// TwinCAT 3 PLC project TestProject
// ProgramVersion: 3.1.4020.4
// libraries:
//   Tc2_EtherCAT, * (Beckhoff Automation GmbH)
//   Tc2_MC2, * (Beckhoff Automation GmbH)
//   Tc2_Standard, * (Beckhoff Automation GmbH)
//   Tc2_System, * (Beckhoff Automation GmbH)
//   Tc3_Module, * (Beckhoff Automation GmbH)
//   tc_mca_std_lib, * (ESS)
// project tree:
//   DUTs/ ST_AxisHardware.TcDUT, ST_AxisParams.TcDUT, ST_EL7031CoEParams.TcDUT
//   / PlcTask.TcTTO
//   POUs/ FB_AxisConfig.TcPOU, FB_AxisEthMaster.TcPOU, FB_AxisHardware.TcPOU, FB_AxisRead5042.TcPOU, FB_AxisRead70x1.TcPOU, FB_AxisReadCoE.TcPOU, FB_AxisReadNC.TcPOU, FB_AxisReadParams.TcPOU, FB_AxisSetSlaveState.TcPOU, FB_AxisWrite5042.TcPOU, FB_AxisWrite70x1.TcPOU, FB_AxisWriteCoE.TcPOU, FB_AxisWriteNC.TcPOU, FB_AxisWriteParams.TcPOU, MAIN.TcPOU, FB_AxisMaster.TcPOU
// real-time tasks:
//   TASK PlcTask: cycle T#10ms, priority 20, ADS port 350
// motion (NC):
//   TASK NC-Task 1 SAF: cycle T#2ms, priority 4, ADS port 501
//   TASK NC-Task 1 SVB: cycle T#10ms, priority 8, ADS port 511
//   AXIS Axis 1 (id 1)
//     OtherSettings: AllowMotionCmdToSlave=true
//     encoder EncType=1
//     drive DrvType=5
//       TimeComp: TaskDelayCycles=1
//     controller CtrType=1
//       CtrPara: PriorControlFactor=1
//         Observer: BandWidth=20
//   AXIS Axis 2 (id 2)
//     OtherSettings: AllowMotionCmdToSlave=true
//     encoder EncType=29
//       EncPara: MaxCount=#xffffffff
//         Inc: RefSoftSyncMask=#x0000ffff
//     drive DrvType=24
//       TimeComp: TaskDelayCycles=1
//     controller CtrType=1
//       CtrPara: PriorControlFactor=1
//         Observer: BandWidth=20
//   AXIS Axis 3 (id 3)
//     OtherSettings: AllowMotionCmdToSlave=true
//     encoder EncType=29
//       EncPara: MaxCount=#xffffffff
//         Inc: RefSoftSyncMask=#x0000ffff
//     drive DrvType=24
//       TimeComp: TaskDelayCycles=1
//     controller CtrType=1
//       CtrPara: PriorControlFactor=1
//         Observer: BandWidth=20
// I/O:
//   DEVICE Device 1 (EtherCAT), AmsNetId 5.45.6.154.2.1
//     Term 1 (EK1200) [EK1200-5000 EtherCAT Power supply (2A E-Bus)]
//       Term 2 (EL7031) [EL7031 1Ch. Stepper motor output stage (24V, 1.5A)]
//       Term 3 (EL7041) [EL7041 1Ch. Stepper motor output stage (50V, 5A)]
//       Term 4 (EL5042) [EL5042 2Ch. BiSS-C Encoder]
//       Term 6 (EL1004) [EL1004 4Ch. Dig. Input 24V, 3ms]
//       Term 7 (EL1004) [EL1004 4Ch. Dig. Input 24V, 3ms]
//       Term 5 (EL9011) [EL9011 End Terminal]
// variable links:
//   (this object) <-> Device 1 (EtherCAT)/Term 1 (EK1200)/Term 2 (EL7031)
//     Drive/Inputs/In/nState1 @bit 3 <-> STM Status/Status/Error
//     Drive/Inputs/In/nState1 @bit 5 <-> STM Status/Status/Moving negative
//     Drive/Inputs/In/nState1 @bit 4 <-> STM Status/Status/Moving positive
//     Drive/Inputs/In/nState1 @bit 1 <-> STM Status/Status/Ready
//     Drive/Inputs/In/nState1 <-> STM Status/Status/Ready to enable
//     Drive/Inputs/In/nState1 @bit 6 <-> STM Status/Status/Torque reduced
//     Drive/Inputs/In/nState1 @bit 2 <-> STM Status/Status/Warning
//     Drive/Inputs/In/nState2 @bit 3 <-> STM Status/Status/Digital input 1
//     Drive/Inputs/In/nState2 @bit 4 <-> STM Status/Status/Digital input 2
//     Drive/Inputs/In/nState2 @bit 5 <-> STM Status/Status/Sync error
//     Drive/Inputs/In/nState2 @bit 7 <-> STM Status/Status/TxPDO Toggle
//     Drive/Inputs/In/nState4 @bit 1 <-> WcState/InputToggle
//     Drive/Inputs/In/nState4 <-> WcState/WcState
//     Drive/Outputs/Out/nCtrl1 <-> STM Control/Control/Enable
//     Drive/Outputs/Out/nCtrl1 @bit 2 <-> STM Control/Control/Reduce torque
//     Drive/Outputs/Out/nCtrl1 @bit 1 <-> STM Control/Control/Reset
//     Drive/Outputs/Out/nDataOut2[0] <-> STM Velocity/Velocity
//   (this object) <-> Device 1 (EtherCAT)/Term 1 (EK1200)/Term 4 (EL5042)
//     Enc/Inputs/In/nComState @bit 1 <-> WcState/InputToggle
//     Enc/Inputs/In/nComState <-> WcState/WcState
//     Enc/Inputs/In/nDataIn1 <-> FB Inputs Channel 1/Position
//     Enc/Inputs/In/nDataIn1 <-> FB Inputs Channel 2/Position
//     Enc/Inputs/In/nState1 @bit 12 <-> FB Inputs Channel 1/Status/Diag
//     Enc/Inputs/In/nState1 @bit 12 <-> FB Inputs Channel 2/Status/Diag
//     Enc/Inputs/In/nState1 @bit 1 <-> FB Inputs Channel 1/Status/Error
//     Enc/Inputs/In/nState1 @bit 1 <-> FB Inputs Channel 2/Status/Error
//     Enc/Inputs/In/nState1 @bit 14 <-> FB Inputs Channel 1/Status/Input cycle counter
//     Enc/Inputs/In/nState1 @bit 14 <-> FB Inputs Channel 2/Status/Input cycle counter
//     Enc/Inputs/In/nState1 @bit 2 <-> FB Inputs Channel 1/Status/Ready
//     Enc/Inputs/In/nState1 @bit 2 <-> FB Inputs Channel 2/Status/Ready
//     Enc/Inputs/In/nState1 @bit 13 <-> FB Inputs Channel 1/Status/TxPDO State
//     Enc/Inputs/In/nState1 @bit 13 <-> FB Inputs Channel 2/Status/TxPDO State
//     Enc/Inputs/In/nState1 <-> FB Inputs Channel 1/Status/Warning
//     Enc/Inputs/In/nState1 <-> FB Inputs Channel 2/Status/Warning
//   (this object) <-> Device 1 (EtherCAT)/Term 1 (EK1200)/Term 3 (EL7041)
//     Drive/Inputs/In/nState1 @bit 3 <-> STM Status/Status/Error
//     Drive/Inputs/In/nState1 @bit 5 <-> STM Status/Status/Moving negative
//     Drive/Inputs/In/nState1 @bit 4 <-> STM Status/Status/Moving positive
//     Drive/Inputs/In/nState1 @bit 1 <-> STM Status/Status/Ready
//     Drive/Inputs/In/nState1 <-> STM Status/Status/Ready to enable
//     Drive/Inputs/In/nState1 @bit 6 <-> STM Status/Status/Torque reduced
//     Drive/Inputs/In/nState1 @bit 2 <-> STM Status/Status/Warning
//     Drive/Inputs/In/nState2 @bit 3 <-> STM Status/Status/Digital input 1
//     Drive/Inputs/In/nState2 @bit 4 <-> STM Status/Status/Digital input 2
//     Drive/Inputs/In/nState4 @bit 1 <-> WcState/InputToggle
//     Drive/Inputs/In/nState4 <-> WcState/WcState
//     Drive/Outputs/Out/nCtrl1 <-> STM Control/Control/Enable
//     Drive/Outputs/Out/nCtrl1 @bit 2 <-> STM Control/Control/Reduce torque
//     Drive/Outputs/Out/nCtrl1 @bit 1 <-> STM Control/Control/Reset
//     Drive/Outputs/Out/nDataOut2[0] <-> STM Velocity/Velocity
//   TestProject Instance <-> Device 1 (EtherCAT)/Term 1 (EK1200)/Term 2 (EL7031)
//     PlcTask Inputs/MAIN.bLimitBwdM2 <-> STM Status/Status/Digital input 2
//     PlcTask Inputs/MAIN.bLimitFwdM2 <-> STM Status/Status/Digital input 1
//   TestProject Instance <-> Device 1 (EtherCAT)/Term 1 (EK1200)/Term 3 (EL7041)
//     PlcTask Inputs/MAIN.bLimitBwdM3 <-> STM Status/Status/Digital input 2
//     PlcTask Inputs/MAIN.bLimitFwdM3 <-> STM Status/Status/Digital input 1
//   TestProject Instance <-> Device 1 (EtherCAT)/Term 1 (EK1200)/Term 4 (EL5042)
//     PlcTask Inputs/MAIN.ams23Enc <-> InfoData/AdsAddr
//   TestProject Instance <-> NC-Task 1 SAF/Axes/Axis 1
//     PlcTask Inputs/MAIN.M1.fbLink.Axis.NcToPlc <-> Outputs/ToPlc
//     PlcTask Outputs/MAIN.M1.fbLink.Axis.PlcToNc <-> Inputs/FromPlc
//   TestProject Instance <-> NC-Task 1 SAF/Axes/Axis 2
//     PlcTask Inputs/MAIN.M2.fbLink.Axis.NcToPlc <-> Outputs/ToPlc
//     PlcTask Outputs/MAIN.M2.fbLink.Axis.PlcToNc <-> Inputs/FromPlc
//   TestProject Instance <-> NC-Task 1 SAF/Axes/Axis 3
//     PlcTask Inputs/MAIN.M3.fbLink.Axis.NcToPlc <-> Outputs/ToPlc
//     PlcTask Outputs/MAIN.M3.fbLink.Axis.PlcToNc <-> Inputs/FromPlc

CONFIGURATION TestProject
    RESOURCE PLC ON TwinCAT3
        TASK PlcTask(INTERVAL := T#10ms, PRIORITY := 20);
        PROGRAM MAIN WITH PlcTask : MAIN;
    END_RESOURCE
END_CONFIGURATION

// ---- DUTs/ST_AxisHardware.TcDUT
TYPE ST_AxisHardware :
STRUCT
	drive_type: UINT;
	enc_type: UINT;
	drive_ref: ST_DriveRef;
	enc_ref: ST_DriveRef;
END_STRUCT
END_TYPE

// ---- DUTs/ST_AxisParams.TcDUT
TYPE ST_AxisParams :
STRUCT
	unit: STRING := 'mm';
	ref_vel: LREAL;
	max_vel: LREAL;
	max_acc: LREAL := 15000;
	max_dec: LREAL := 15000;
	def_acc: LREAL := 1500;
	def_dec: LREAL := 1500;
	def_jerk: LREAL := 2250;
	home_search: LREAL;
	home_sync: LREAL;
	man_fast: LREAL;
	man_slow: LREAL;
	enable_min_soft_limit: BOOL;
	enable_max_soft_limit: BOOL;
	min_soft_limit: LREAL;
	max_soft_limit: LREAL;
	max_pos_lag_value: LREAL := 5;
	max_pos_lag_filter_time: LREAL := 0.02;
	dead_time: LREAL := 0.008;
	enc_scale: LREAL;
	enc_offset: LREAL;
	enc_invert: BOOL;
	mot_invert: BOOL;
	max_current: UINT;
	holding_current: UINT := 100;
	voltage: UINT := 24000;
	resistance: UINT := 100;
	emf: UINT := 0;
	full_steps: UINT := 200;
	speed_range: USINT := 1;
	enc_supply: USINT := 50;
	enc_clock: USINT := 9;
	enc_multi_bits: USINT := 0;
	enc_single_bits: USINT := 32;
END_STRUCT
END_TYPE

// ---- DUTs/ST_EL7031CoEParams.TcDUT
TYPE ST_EL7031CoEParams :
STRUCT
END_STRUCT
END_TYPE

// ---- POUs/MAIN.TcPOU
PROGRAM MAIN
VAR
	fbAxisEthMaster: FB_AxisEthMaster;
	M1: FB_AxisMaster;
	M2: FB_AxisMaster;
	M3: FB_AxisMaster;
	bFirstCycle: BOOL := TRUE;
END_VAR

// Set the initial configs
IF bFirstCycle THEN
	M2.stConfigSet.ref_vel := 10;
	M2.stConfigSet.max_vel := 20;
	M2.stConfigSet.man_fast := 15;
	M2.stConfigSet.man_slow := 5;
	M2.stConfigSet.enc_scale := 0.001;
	M2.stConfigSet.max_current := 1100;
	M3.stConfigSet.ref_vel := 11;
	M3.stConfigSet.max_vel := 21;
	M3.stConfigSet.man_fast := 16;
	M3.stConfigSet.man_slow := 6;
	M3.stConfigSet.enc_scale := 0.002;
	M3.stConfigSet.max_current := 1234;
	bFirstCycle := FALSE;
END_IF

// Bring MASTER to OP once SLAVEs are PRE-OP
fbAxisEthMaster(bExecute:=M1.bInitPreOp AND M2.bInitPreOp AND M3.bInitPreOp);

// Enable and pass Cfg
M1(bEnable:=TRUE,
	bInitCfg:=FALSE,
	bCfgRO:=FALSE,
	bUseLimits:=FALSE);
M2(bEnable:=TRUE,
	bInitCfg:=TRUE,
	bCfgRO:=FALSE,
	nEncCh:=1);
M3(bEnable:=TRUE,
	bInitCfg:=TRUE,
	bCfgRO:=TRUE,
	nEncCh:=2);

END_PROGRAM

// ---- POUs/FB_AxisEthMaster.TcPOU
FUNCTION_BLOCK FB_AxisEthMaster
VAR_INPUT
	bExecute: BOOL := TRUE;
END_VAR
VAR_OUTPUT
	bCfgReady: BOOL;
END_VAR
VAR
	amsNetID AT %I*: AMSNETID;
	fbMasterOp: FB_EcSetMasterState;
END_VAR

// Set master to OP
// This should wait until all relevant slaves are set to PREOP or they will be prematurely set to OP
fbMasterOp(sNetId:=F_CREATEAMSNETID(amsNetID),
	bExecute:=bExecute,
	reqState:=EC_DEVICE_STATE_OP);

END_FUNCTION_BLOCK

// ---- POUs/FB_AxisMaster.TcPOU
FUNCTION_BLOCK FB_AxisMaster
VAR_INPUT
	bEnable: BOOL;
	bInitCfg: BOOL := TRUE;
	bCfgRO: BOOL := FALSE;
	bUseLimits: BOOL;
	nEncCh: USINT;
END_VAR
VAR_OUTPUT
	bBrakeOut AT %I*: BOOL;
	bInitPreOp: BOOL;
	stConfigGet: ST_AxisParams;
END_VAR
VAR
	stConfigSet: ST_AxisParams;
	bLimitFwd AT %I*: BOOL;
	bLimitBwd AT %I*: BOOL;
	bHomeSensor AT %I*: BOOL;
	amsEncAddr AT %I*: AMSADDR;
	fbLink: FB_NcAxis;
	fbHardware: FB_AxisHardware;
	fbConfig: FB_AxisConfig;
	fbMasterGetOP: FB_EcGetMasterState;
	fbAxisSetOP: FB_AxisSetSlaveState;
	fbDrive: FB_DriveVirtual;
	stAxisStatus: DUT_AxisStatus_v0_01;
	bExecConfig: BOOL;
END_VAR

// Landing zone to link the AXIS_REF and update it
fbLink(En:=bEnable);
// Get terminal info
fbHardware(bExecute:=bEnable,
	Axis:=fbLink.Axis,
	amsEncAddr:=amsEncAddr,
	nEncCh:=nEncCh);
// If asked to initialize and we haven't, then initialize
IF bInitCfg AND NOT fbConfig.bInitDone THEN
	bExecConfig := TRUE;
// If read-only and not initializing, reject the write command
ELSIF bCfgRO THEN
	bExecConfig := FALSE;
// Otherwise, keep the value written over ADS
END_IF
// Read and/or write the config
fbConfig(bExecute:=bExecConfig AND fbHardware.bDone,
	stConfigSet:=stConfigSet,
	stHardware:=fbHardware.stHardware,
	Axis:=fbLink.Axis,
	bInitPreOp=>bInitPreOp,
	stConfigGet=>stConfigGet);
// Reset the execute bool
IF fbConfig.bDone AND NOT fbConfig.bError THEN
	bExecConfig := FALSE;
END_IF
// After the initial config is done, go to OP mode
// But first, make sure the master is in OP mode
IF fbConfig.bDone AND NOT fbConfig.bError AND fbMasterGetOP.state <> EC_DEVICE_STATE_OP THEN
	IF fbMasterGetOP.bExecute AND NOT fbMasterGetOP.bBusy THEN
		fbMasterGetOP.bExecute := FALSE;
	ELSE
		fbMasterGetOP.bExecute := TRUE;
	END_IF
END_IF
fbMasterGetOP(sNetId:=fbHardware.stHardware.drive_ref.sNetId);
fbAxisSetOP(bExecute:=fbConfig.bDone AND NOT fbConfig.bError,
	stHardware:=fbHardware.stHardware,
	reqState:=EC_DEVICE_STATE_OP);

// Disable brake while executing move **TODO** make this robust
bBrakeOut := fbDrive.bExecute;

IF NOT bUseLimits THEN
	bLimitFwd := TRUE;
	bLimitBwd := TRUE;
END_IF
// Execute incoming motion commands
fbDrive(En:=bEnable,
	bEnable:=bEnable AND fbConfig.bInitDone,
	bLimitFwd:=bLimitFwd,
	bLimitBwd:=bLimitBwd,
	bHomeSensor:=bHomeSensor,
	Axis:=fbLink.Axis);
stAxisStatus := fbDrive.stAxisStatus;
// Reset the execute bool
IF fbDrive.bDone AND NOT fbDrive.bError THEN
	fbDrive.bExecute := FALSE;
END_IF

END_FUNCTION_BLOCK

// ---- POUs/FB_AxisHardware.TcPOU
FUNCTION_BLOCK FB_AxisHardware
VAR_INPUT
	bExecute: BOOL;
	amsEncAddr: AMSADDR;
	nEncCh: USINT;
END_VAR
VAR_IN_OUT
	Axis: AXIS_REF;
END_VAR
VAR_OUTPUT
	bDone: BOOL;
	bBusy: BOOL;
	bError: BOOL;
	nErrorID: UDINT;
	stHardware: ST_AxisHardware;
END_VAR
VAR
	fbReadDriveAddress: MC_ReadDriveAddress;
	fbDriveId: FB_EcGetSlaveIdentity;
	fbEncId: FB_EcGetSlaveIdentity;
	fbADSRead: ADSREADEX;
	stDriveAddr: ST_DriveAddress;
	stDriveRef: ST_DriveRef;
	stEncRef: ST_DriveRef;
END_VAR

// Get drive ref using AXIS_REF
fbReadDriveAddress(Execute:=bExecute,
	Axis:=Axis,
	DriveAddress=>stDriveAddr);
stDriveRef.sNetId := stDriveAddr.NetID;
stDriveRef.nSlaveAddr := stDriveAddr.SlaveAddress;
stDriveRef.nDriveNo := stDriveAddr.Channel;
stHardware.drive_ref := stDriveRef;

// Get encoder ref using input args (cannot be derived from AXIS_REF)
stEncRef.sNetId := F_CreateAmsNetId(amsEncAddr.netId);
stEncRef.nSlaveAddr := amsEncAddr.port;
stEncRef.nDriveNo := nEncCh;
stHardware.enc_ref := stEncRef;

// Get the drive model (e.g. 7031)
IF stDriveRef.nSlaveAddr > 0 THEN
	fbDriveId(bExecute:=bExecute AND fbReadDriveAddress.Done,
		sNetId:=stDriveRef.sNetId,
		nSlaveAddr:=stDriveRef.nSlaveAddr);
	stHardware.drive_type := UDINT_TO_UINT(SHR(fbDriveID.identity.productCode, 16));
END_IF

// Get the encoder model (e.g. 5042)
IF stEncRef.nSlaveAddr > 0 THEN
	fbEncId(bExecute:=bExecute AND fbReadDriveAddress.Done,
		sNetId:=stEncRef.sNetId,
		nSlaveAddr:=stEncRef.nSlaveAddr);
	stHardware.enc_type := UDINT_TO_UINT(SHR(fbEncID.identity.productCode, 16));
END_IF

// Summarize outputs
bDone := fbReadDriveAddress.Done AND NOT fbDriveId.bBusy AND NOT fbEncId.bBusy;
bBusy := fbReadDriveAddress.Busy OR fbDriveId.bBusy OR fbEncId.bBusy;
bError := fbReadDriveAddress.Error OR fbDriveId.bError OR fbEncId.bError;
IF fbReadDriveAddress.ErrorID > 0 THEN
	nErrorID := fbReadDriveAddress.ErrorID;
ELSIF fbDriveId.nErrId >0 THEN
	nErrorID := fbDriveId.nErrId;
ELSE
	nErrorID := fbEncId.nErrId;
END_IF

END_FUNCTION_BLOCK

// ---- POUs/FB_AxisConfig.TcPOU
FUNCTION_BLOCK FB_AxisConfig
VAR_INPUT
	bExecute: BOOL; // Set, then get
	bExecGet: BOOL; // Only get
	bReset: BOOL;
	stConfigSet: ST_AxisParams;
	stHardware: ST_AxisHardware;
END_VAR
VAR_IN_OUT
	Axis: AXIS_REF;
END_VAR
VAR_OUTPUT
	bDone: BOOL;
	bValid: BOOL;
	bBusy: BOOL;
	bError: BOOL;
	nErrorID: UDINT;
	bInitDone: BOOL;
	bInitPreOp: BOOL;
	stConfigGet: ST_AxisParams;
END_VAR
VAR
	fbRead: FB_AxisReadParams;
	fbWrite: FB_AxisWriteParams;
	bDoRead: BOOL;
END_VAR

// Write first
fbWrite(bExecute:=bExecute,
	bReset:=bReset,
	stConfig:=stConfigSet,
	stHardware:=stHardware,
	Axis:=Axis,
	bInitPreOp=>bInitPreOp);
// Reset bDoRead if both execs are false
IF NOT bExecute AND NOT bExecGet THEN
	bDoRead := FALSE;
END_IF
// If bExecute is TRUE, wait untill after the write to read
IF bExecute THEN
	bDoRead := fbWrite.bDone;
ELSE
	bDoRead := bExecGet;
END_IF
// Notify that its ok to set master to OP.
// This block is really only used if we skip the write step.
IF bDoRead THEN
	bInitPreOP := TRUE;
END_IF
// Read now
fbRead(bExecute:=bDoRead,
	bReset:=bReset,
	stHardware:=stHardware,
	Axis:=Axis,
	stConfig=>stConfigGet,
	bValid=>bValid);
// Set the status outputs
bDone := fbWrite.bDone AND NOT fbRead.bBusy;
bBusy := fbWrite.bBusy OR fbRead.bBusy;
bError := fbWrite.bError OR fbRead.bError;
IF fbWrite.nErrorID > 0 THEN
	nErrorID := fbWrite.nErrorID;
ELSE
	nErrorID := fbRead.nErrorID;
END_IF
IF bDone THEN
	bInitDone := TRUE;
END_IF
IF bError THEN
	bInitDone := FALSE;
END_IF

END_FUNCTION_BLOCK

// ---- POUs/FB_AxisReadParams.TcPOU
FUNCTION_BLOCK FB_AxisReadParams
VAR_INPUT
	bExecute: BOOL;
	bReset: BOOL;
	stHardware: ST_AxisHardware;
END_VAR
VAR_OUTPUT
	stConfig: ST_AxisParams;
	bValid: BOOL;
	bBusy: BOOL;
	bError: BOOL;
	nErrorID: UDINT;
END_VAR
VAR_IN_OUT
	Axis: AXIS_REF;
END_VAR
VAR
	fbNCRead: FB_AxisReadNC;
	fbCoERead: FB_AxisReadCoE;
END_VAR

fbNCRead(bExecute:=bExecute,
	bReset:=bReset,
	stConfig:=stConfig,
	Axis:=Axis);
fbCoERead(bExecute:=bExecute,
	bReset:=bReset,
	stHardware:=stHardware,
	stConfig:=stConfig,
	Axis:=Axis);
bValid := fbNCRead.bValid AND NOT fbCoERead.bBusy AND NOT fbCoERead.bError AND bExecute;
bBusy := fbNCRead.bBusy OR fbCoERead.bBusy;
bError := fbNCRead.bError OR fbCoERead.bError;
IF fbNCRead.nErrorID > 0 THEN
	nErrorID := fbNCRead.nErrorID;
ELSE
	nErrorID := fbCoERead.nErrorID;
END_IF

END_FUNCTION_BLOCK

// ---- POUs/FB_AxisReadNC.TcPOU
FUNCTION_BLOCK FB_AxisReadNC
VAR_INPUT
	bExecute: BOOL;
	bReset: BOOL;
END_VAR
VAR_IN_OUT
	stConfig: ST_AxisParams;
	Axis: AXIS_REF;
END_VAR
VAR_OUTPUT
	bValid: BOOL;
	bBusy: BOOL;
	bError: BOOL;
	nErrorID: UDINT;
END_VAR
VAR
	fbReadRefVel: MC_ReadParameter;
  	fbReadRefVelRisingEdge: R_TRIG;
	fbReadMaxVel: MC_ReadParameter;
  	fbReadMaxVelRisingEdge: R_TRIG;
	fbReadMaxAcc: MC_ReadParameter;
  	fbReadMaxAccRisingEdge: R_TRIG;
	fbReadMaxDec: MC_ReadParameter;
  	fbReadMaxDecRisingEdge: R_TRIG;
	fbReadDefAcc: MC_ReadParameter;
  	fbReadDefAccRisingEdge: R_TRIG;
	fbReadDefDec: MC_ReadParameter;
  	fbReadDefDecRisingEdge: R_TRIG;
	fbReadDefJerk: MC_ReadParameter;
  	fbReadDefJerkRisingEdge: R_TRIG;
	fbReadHomeSearch: MC_ReadParameter;
  	fbReadHomeSearchRisingEdge: R_TRIG;
	fbReadHomeSync: MC_ReadParameter;
  	fbReadHomeSyncRisingEdge: R_TRIG;
	fbReadManFast: MC_ReadParameter;
  	fbReadManFastRisingEdge: R_TRIG;
	fbReadManSlow: MC_ReadParameter;
  	fbReadManSlowRisingEdge: R_TRIG;
	fbReadEnableMinSoftLimit: MC_ReadBoolParameter;
  	fbReadEnableMinSoftLimitRisingEdge: R_TRIG;
	fbReadEnableMaxSoftLimit: MC_ReadBoolParameter;
  	fbReadEnableMaxSoftLimitRisingEdge: R_TRIG;
	fbReadMinSoftLimit: MC_ReadParameter;
  	fbReadMinSoftLimitRisingEdge: R_TRIG;
	fbReadMaxSoftLimit: MC_ReadParameter;
  	fbReadMaxSoftLimitRisingEdge: R_TRIG;
	fbReadMaxPosLagValue: MC_ReadParameter;
  	fbReadMaxPosLagValueRisingEdge: R_TRIG;
	fbReadMaxPosLagFilterTime: MC_ReadParameter;
  	fbReadMaxPosLagFilterTimeRisingEdge: R_TRIG;
	fbReadDeadTime: MC_ReadParameter;
  	fbReadDeadTimeRisingEdge: R_TRIG;
	fbReadEncScale: MC_ReadParameter;
  	fbReadEncScaleRisingEdge: R_TRIG;
	fbReadEncOffset: MC_ReadParameter;
  	fbReadEncOffsetRisingEdge: R_TRIG;
	fbReadEncInvert: MC_ReadBoolParameter;
  	fbReadEncInvertRisingEdge: R_TRIG;
	fbReadMotInvert: MC_ReadBoolParameter;
  	fbReadMotInvertRisingEdge: R_TRIG;
END_VAR

// File auto-generated! Take care editing!
// Clears errors and allows a new read
IF bReset THEN
	bExecute := FALSE;
	bReset := FALSE;
END_IF
fbReadRefVel(Enable:=bExecute,
	ParameterNumber:=MC_AxisParameter.AxisRefVeloOnRefOutput,
	ReadMode:=E_ReadMode.READMODE_ONCE,
	Axis:=Axis);
fbReadRefVelRisingEdge(CLK:=fbReadRefVel.Valid AND NOT fbReadRefVel.Busy);
IF fbReadRefVelRisingEdge.Q AND NOT fbReadRefVel.Error THEN
	stConfig.ref_vel := fbReadRefVel.Value;
END_IF
fbReadMaxVel(Enable:=bExecute,
	ParameterNumber:=MC_AxisParameter.AxisMaxVelocity,
	ReadMode:=E_ReadMode.READMODE_ONCE,
	Axis:=Axis);
fbReadMaxVelRisingEdge(CLK:=fbReadMaxVel.Valid AND NOT fbReadMaxVel.Busy);
IF fbReadMaxVelRisingEdge.Q AND NOT fbReadMaxVel.Error THEN
	stConfig.max_vel := fbReadMaxVel.Value;
END_IF
fbReadMaxAcc(Enable:=bExecute,
	ParameterNumber:=MC_AxisParameter.MaxAccelerationSystem,
	ReadMode:=E_ReadMode.READMODE_ONCE,
	Axis:=Axis);
fbReadMaxAccRisingEdge(CLK:=fbReadMaxAcc.Valid AND NOT fbReadMaxAcc.Busy);
IF fbReadMaxAccRisingEdge.Q AND NOT fbReadMaxAcc.Error THEN
	stConfig.max_acc := fbReadMaxAcc.Value;
END_IF
fbReadMaxDec(Enable:=bExecute,
	ParameterNumber:=MC_AxisParameter.MaxDecelerationSystem,
	ReadMode:=E_ReadMode.READMODE_ONCE,
	Axis:=Axis);
fbReadMaxDecRisingEdge(CLK:=fbReadMaxDec.Valid AND NOT fbReadMaxDec.Busy);
IF fbReadMaxDecRisingEdge.Q AND NOT fbReadMaxDec.Error THEN
	stConfig.max_dec := fbReadMaxDec.Value;
END_IF
fbReadDefAcc(Enable:=bExecute,
	ParameterNumber:=MC_AxisParameter.AxisAcc,
	ReadMode:=E_ReadMode.READMODE_ONCE,
	Axis:=Axis);
fbReadDefAccRisingEdge(CLK:=fbReadDefAcc.Valid AND NOT fbReadDefAcc.Busy);
IF fbReadDefAccRisingEdge.Q AND NOT fbReadDefAcc.Error THEN
	stConfig.def_acc := fbReadDefAcc.Value;
END_IF
fbReadDefDec(Enable:=bExecute,
	ParameterNumber:=MC_AxisParameter.AxisDec,
	ReadMode:=E_ReadMode.READMODE_ONCE,
	Axis:=Axis);
fbReadDefDecRisingEdge(CLK:=fbReadDefDec.Valid AND NOT fbReadDefDec.Busy);
IF fbReadDefDecRisingEdge.Q AND NOT fbReadDefDec.Error THEN
	stConfig.def_dec := fbReadDefDec.Value;
END_IF
fbReadDefJerk(Enable:=bExecute,
	ParameterNumber:=MC_AxisParameter.AxisJerk,
	ReadMode:=E_ReadMode.READMODE_ONCE,
	Axis:=Axis);
fbReadDefJerkRisingEdge(CLK:=fbReadDefJerk.Valid AND NOT fbReadDefJerk.Busy);
IF fbReadDefJerkRisingEdge.Q AND NOT fbReadDefJerk.Error THEN
	stConfig.def_jerk := fbReadDefJerk.Value;
END_IF
fbReadHomeSearch(Enable:=bExecute,
	ParameterNumber:=MC_AxisParameter.AxisCalibrationVelocityForward,
	ReadMode:=E_ReadMode.READMODE_ONCE,
	Axis:=Axis);
fbReadHomeSearchRisingEdge(CLK:=fbReadHomeSearch.Valid AND NOT fbReadHomeSearch.Busy);
IF fbReadHomeSearchRisingEdge.Q AND NOT fbReadHomeSearch.Error THEN
	stConfig.home_search := fbReadHomeSearch.Value;
END_IF
fbReadHomeSync(Enable:=bExecute,
	ParameterNumber:=MC_AxisParameter.AxisCalibrationVelocityBackward,
	ReadMode:=E_ReadMode.READMODE_ONCE,
	Axis:=Axis);
fbReadHomeSyncRisingEdge(CLK:=fbReadHomeSync.Valid AND NOT fbReadHomeSync.Busy);
IF fbReadHomeSyncRisingEdge.Q AND NOT fbReadHomeSync.Error THEN
	stConfig.home_sync := fbReadHomeSync.Value;
END_IF
fbReadManFast(Enable:=bExecute,
	ParameterNumber:=MC_AxisParameter.AxisManualVelocityFast,
	ReadMode:=E_ReadMode.READMODE_ONCE,
	Axis:=Axis);
fbReadManFastRisingEdge(CLK:=fbReadManFast.Valid AND NOT fbReadManFast.Busy);
IF fbReadManFastRisingEdge.Q AND NOT fbReadManFast.Error THEN
	stConfig.man_fast := fbReadManFast.Value;
END_IF
fbReadManSlow(Enable:=bExecute,
	ParameterNumber:=MC_AxisParameter.AxisManualVelocitySlow,
	ReadMode:=E_ReadMode.READMODE_ONCE,
	Axis:=Axis);
fbReadManSlowRisingEdge(CLK:=fbReadManSlow.Valid AND NOT fbReadManSlow.Busy);
IF fbReadManSlowRisingEdge.Q AND NOT fbReadManSlow.Error THEN
	stConfig.man_slow := fbReadManSlow.Value;
END_IF
fbReadEnableMinSoftLimit(Enable:=bExecute,
	ParameterNumber:=MC_AxisParameter.EnableLimitNeg,
	ReadMode:=E_ReadMode.READMODE_ONCE,
	Axis:=Axis);
fbReadEnableMinSoftLimitRisingEdge(CLK:=fbReadEnableMinSoftLimit.Valid AND NOT fbReadEnableMinSoftLimit.Busy);
IF fbReadEnableMinSoftLimitRisingEdge.Q AND NOT fbReadEnableMinSoftLimit.Error THEN
	stConfig.enable_min_soft_limit := fbReadEnableMinSoftLimit.Value;
END_IF
fbReadEnableMaxSoftLimit(Enable:=bExecute,
	ParameterNumber:=MC_AxisParameter.EnableLimitPos,
	ReadMode:=E_ReadMode.READMODE_ONCE,
	Axis:=Axis);
fbReadEnableMaxSoftLimitRisingEdge(CLK:=fbReadEnableMaxSoftLimit.Valid AND NOT fbReadEnableMaxSoftLimit.Busy);
IF fbReadEnableMaxSoftLimitRisingEdge.Q AND NOT fbReadEnableMaxSoftLimit.Error THEN
	stConfig.enable_max_soft_limit := fbReadEnableMaxSoftLimit.Value;
END_IF
fbReadMinSoftLimit(Enable:=bExecute,
	ParameterNumber:=MC_AxisParameter.SWLimitNeg,
	ReadMode:=E_ReadMode.READMODE_ONCE,
	Axis:=Axis);
fbReadMinSoftLimitRisingEdge(CLK:=fbReadMinSoftLimit.Valid AND NOT fbReadMinSoftLimit.Busy);
IF fbReadMinSoftLimitRisingEdge.Q AND NOT fbReadMinSoftLimit.Error THEN
	stConfig.min_soft_limit := fbReadMinSoftLimit.Value;
END_IF
fbReadMaxSoftLimit(Enable:=bExecute,
	ParameterNumber:=MC_AxisParameter.SWLimitPos,
	ReadMode:=E_ReadMode.READMODE_ONCE,
	Axis:=Axis);
fbReadMaxSoftLimitRisingEdge(CLK:=fbReadMaxSoftLimit.Valid AND NOT fbReadMaxSoftLimit.Busy);
IF fbReadMaxSoftLimitRisingEdge.Q AND NOT fbReadMaxSoftLimit.Error THEN
	stConfig.max_soft_limit := fbReadMaxSoftLimit.Value;
END_IF
fbReadMaxPosLagValue(Enable:=bExecute,
	ParameterNumber:=MC_AxisParameter.MaxPositionLag,
	ReadMode:=E_ReadMode.READMODE_ONCE,
	Axis:=Axis);
fbReadMaxPosLagValueRisingEdge(CLK:=fbReadMaxPosLagValue.Valid AND NOT fbReadMaxPosLagValue.Busy);
IF fbReadMaxPosLagValueRisingEdge.Q AND NOT fbReadMaxPosLagValue.Error THEN
	stConfig.max_pos_lag_value := fbReadMaxPosLagValue.Value;
END_IF
fbReadMaxPosLagFilterTime(Enable:=bExecute,
	ParameterNumber:=MC_AxisParameter.AxisMaxPosLagFilterTime,
	ReadMode:=E_ReadMode.READMODE_ONCE,
	Axis:=Axis);
fbReadMaxPosLagFilterTimeRisingEdge(CLK:=fbReadMaxPosLagFilterTime.Valid AND NOT fbReadMaxPosLagFilterTime.Busy);
IF fbReadMaxPosLagFilterTimeRisingEdge.Q AND NOT fbReadMaxPosLagFilterTime.Error THEN
	stConfig.max_pos_lag_filter_time := fbReadMaxPosLagFilterTime.Value;
END_IF
fbReadDeadTime(Enable:=bExecute,
	ParameterNumber:=MC_AxisParameter.AxisDelayTimeVeloPosition,
	ReadMode:=E_ReadMode.READMODE_ONCE,
	Axis:=Axis);
fbReadDeadTimeRisingEdge(CLK:=fbReadDeadTime.Valid AND NOT fbReadDeadTime.Busy);
IF fbReadDeadTimeRisingEdge.Q AND NOT fbReadDeadTime.Error THEN
	stConfig.dead_time := fbReadDeadTime.Value;
END_IF
fbReadEncScale(Enable:=bExecute,
	ParameterNumber:=MC_AxisParameter.AxisEncoderScalingFactor,
	ReadMode:=E_ReadMode.READMODE_ONCE,
	Axis:=Axis);
fbReadEncScaleRisingEdge(CLK:=fbReadEncScale.Valid AND NOT fbReadEncScale.Busy);
IF fbReadEncScaleRisingEdge.Q AND NOT fbReadEncScale.Error THEN
	stConfig.enc_scale := fbReadEncScale.Value;
END_IF
fbReadEncOffset(Enable:=bExecute,
	ParameterNumber:=MC_AxisParameter.AxisEncoderOffset,
	ReadMode:=E_ReadMode.READMODE_ONCE,
	Axis:=Axis);
fbReadEncOffsetRisingEdge(CLK:=fbReadEncOffset.Valid AND NOT fbReadEncOffset.Busy);
IF fbReadEncOffsetRisingEdge.Q AND NOT fbReadEncOffset.Error THEN
	stConfig.enc_offset := fbReadEncOffset.Value;
END_IF
fbReadEncInvert(Enable:=bExecute,
	ParameterNumber:=MC_AxisParameter.AxisEncoderDirectionInverse,
	ReadMode:=E_ReadMode.READMODE_ONCE,
	Axis:=Axis);
fbReadEncInvertRisingEdge(CLK:=fbReadEncInvert.Valid AND NOT fbReadEncInvert.Busy);
IF fbReadEncInvertRisingEdge.Q AND NOT fbReadEncInvert.Error THEN
	stConfig.enc_invert := fbReadEncInvert.Value;
END_IF
fbReadMotInvert(Enable:=bExecute,
	ParameterNumber:=MC_AxisParameter.AxisMotorDirectionInverse,
	ReadMode:=E_ReadMode.READMODE_ONCE,
	Axis:=Axis);
fbReadMotInvertRisingEdge(CLK:=fbReadMotInvert.Valid AND NOT fbReadMotInvert.Busy);
IF fbReadMotInvertRisingEdge.Q AND NOT fbReadMotInvert.Error THEN
	stConfig.mot_invert := fbReadMotInvert.Value;
END_IF
bValid := fbReadRefVel.Valid AND fbReadMaxVel.Valid AND fbReadMaxAcc.Valid AND fbReadMaxDec.Valid AND fbReadDefAcc.Valid AND fbReadDefDec.Valid AND fbReadDefJerk.Valid AND fbReadHomeSearch.Valid AND fbReadHomeSync.Valid AND fbReadManFast.Valid AND fbReadManSlow.Valid AND fbReadEnableMinSoftLimit.Valid AND fbReadEnableMaxSoftLimit.Valid AND fbReadMinSoftLimit.Valid AND fbReadMaxSoftLimit.Valid AND fbReadMaxPosLagValue.Valid AND fbReadMaxPosLagFilterTime.Valid AND fbReadDeadTime.Valid AND fbReadEncScale.Valid AND fbReadEncOffset.Valid AND fbReadEncInvert.Valid AND fbReadMotInvert.Valid;
bBusy := fbReadRefVel.Busy OR fbReadMaxVel.Busy OR fbReadMaxAcc.Busy OR fbReadMaxDec.Busy OR fbReadDefAcc.Busy OR fbReadDefDec.Busy OR fbReadDefJerk.Busy OR fbReadHomeSearch.Busy OR fbReadHomeSync.Busy OR fbReadManFast.Busy OR fbReadManSlow.Busy OR fbReadEnableMinSoftLimit.Busy OR fbReadEnableMaxSoftLimit.Busy OR fbReadMinSoftLimit.Busy OR fbReadMaxSoftLimit.Busy OR fbReadMaxPosLagValue.Busy OR fbReadMaxPosLagFilterTime.Busy OR fbReadDeadTime.Busy OR fbReadEncScale.Busy OR fbReadEncOffset.Busy OR fbReadEncInvert.Busy OR fbReadMotInvert.Busy;
bError := fbReadRefVel.Error OR fbReadMaxVel.Error OR fbReadMaxAcc.Error OR fbReadMaxDec.Error OR fbReadDefAcc.Error OR fbReadDefDec.Error OR fbReadDefJerk.Error OR fbReadHomeSearch.Error OR fbReadHomeSync.Error OR fbReadManFast.Error OR fbReadManSlow.Error OR fbReadEnableMinSoftLimit.Error OR fbReadEnableMaxSoftLimit.Error OR fbReadMinSoftLimit.Error OR fbReadMaxSoftLimit.Error OR fbReadMaxPosLagValue.Error OR fbReadMaxPosLagFilterTime.Error OR fbReadDeadTime.Error OR fbReadEncScale.Error OR fbReadEncOffset.Error OR fbReadEncInvert.Error OR fbReadMotInvert.Error;
IF NOT bError THEN
	nErrorID := 0;
ELSIF fbReadRefVel.ErrorID > 0 THEN
	nErrorID := fbReadRefVel.ErrorID;
ELSIF fbReadMaxVel.ErrorID > 0 THEN
	nErrorID := fbReadMaxVel.ErrorID;
ELSIF fbReadMaxAcc.ErrorID > 0 THEN
	nErrorID := fbReadMaxAcc.ErrorID;
ELSIF fbReadMaxDec.ErrorID > 0 THEN
	nErrorID := fbReadMaxDec.ErrorID;
ELSIF fbReadDefAcc.ErrorID > 0 THEN
	nErrorID := fbReadDefAcc.ErrorID;
ELSIF fbReadDefDec.ErrorID > 0 THEN
	nErrorID := fbReadDefDec.ErrorID;
ELSIF fbReadDefJerk.ErrorID > 0 THEN
	nErrorID := fbReadDefJerk.ErrorID;
ELSIF fbReadHomeSearch.ErrorID > 0 THEN
	nErrorID := fbReadHomeSearch.ErrorID;
ELSIF fbReadHomeSync.ErrorID > 0 THEN
	nErrorID := fbReadHomeSync.ErrorID;
ELSIF fbReadManFast.ErrorID > 0 THEN
	nErrorID := fbReadManFast.ErrorID;
ELSIF fbReadManSlow.ErrorID > 0 THEN
	nErrorID := fbReadManSlow.ErrorID;
ELSIF fbReadEnableMinSoftLimit.ErrorID > 0 THEN
	nErrorID := fbReadEnableMinSoftLimit.ErrorID;
ELSIF fbReadEnableMaxSoftLimit.ErrorID > 0 THEN
	nErrorID := fbReadEnableMaxSoftLimit.ErrorID;
ELSIF fbReadMinSoftLimit.ErrorID > 0 THEN
	nErrorID := fbReadMinSoftLimit.ErrorID;
ELSIF fbReadMaxSoftLimit.ErrorID > 0 THEN
	nErrorID := fbReadMaxSoftLimit.ErrorID;
ELSIF fbReadMaxPosLagValue.ErrorID > 0 THEN
	nErrorID := fbReadMaxPosLagValue.ErrorID;
ELSIF fbReadMaxPosLagFilterTime.ErrorID > 0 THEN
	nErrorID := fbReadMaxPosLagFilterTime.ErrorID;
ELSIF fbReadDeadTime.ErrorID > 0 THEN
	nErrorID := fbReadDeadTime.ErrorID;
ELSIF fbReadEncScale.ErrorID > 0 THEN
	nErrorID := fbReadEncScale.ErrorID;
ELSIF fbReadEncOffset.ErrorID > 0 THEN
	nErrorID := fbReadEncOffset.ErrorID;
ELSIF fbReadEncInvert.ErrorID > 0 THEN
	nErrorID := fbReadEncInvert.ErrorID;
ELSIF fbReadMotInvert.ErrorID > 0 THEN
	nErrorID := fbReadMotInvert.ErrorID;
END_IF

END_FUNCTION_BLOCK

// ---- POUs/FB_AxisReadCoE.TcPOU
FUNCTION_BLOCK FB_AxisReadCoE
VAR_INPUT
	bExecute: BOOL;
	bReset: BOOL;
	stHardware: ST_AxisHardware;
END_VAR
VAR_IN_OUT
	stConfig: ST_AxisParams;
	Axis: AXIS_REF;
END_VAR
VAR_OUTPUT
	bBusy: BOOL;
	bError: BOOL;
	nErrorID: UDINT;
END_VAR
VAR
	fbRead70x1: FB_AxisRead70x1;
	fbRead5042: FB_AxisRead5042;
	bBusyDrive: BOOL;
	bBusyEnc: BOOL;
	bErrorDrive: BOOL;
	bErrorEnc: BOOL;
	iErrorDriveADS: UDINT;
	iErrorEncADS: UDINT;
	iErrorDriveCAN: UDINT;
	iErrorEncCAN: UDINT;
END_VAR

CASE stHardware.drive_type OF
	0:
		bBusyDrive := FALSE;
		bErrorDrive := FALSE;
		iErrorDriveAds := 0;
		iErrorDriveCAN := 0;
	7031, 7041:
		fbRead70x1(bExecute:=bExecute,
			bReset:=bReset,
			stDriveRef:=stHardware.drive_ref,
			stConfig:=stConfig,
			Axis:=Axis,
			bBusy=>bBusyDrive,
			bError=>bErrorDrive,
			iAdsErrId=>iErrorDriveAds,
			iCANopenErrId=>iErrorDriveCAN);
	ELSE
		bBusyDrive := FALSE;
		bErrorDrive := TRUE;
		iErrorDriveAds := 1;
		iErrorDriveCAN := 0;
END_CASE
CASE stHardware.enc_type OF
	0:
		bBusyEnc := FALSE;
		bErrorEnc := FALSE;
		iErrorEncAds := 0;
		iErrorEncCAN := 0;
	5042:
		fbRead5042(bExecute:=bExecute,
			bReset:=bReset,
			stDriveRef:=stHardware.enc_ref,
			stConfig:=stConfig,
			Axis:=Axis,
			bBusy=>bBusyEnc,
			bError=>bErrorEnc,
			iAdsErrId=>iErrorEncAds,
			iCANopenErrId=>iErrorEncCAN);
	ELSE
		bBusyEnc := FALSE;
		bErrorEnc := TRUE;
		iErrorEncAds := 1;
		iErrorEncCAN := 0;
END_CASE
bBusy := bBusyDrive OR bBusyEnc;
bError := bErrorDrive OR bErrorEnc;
IF iErrorDriveAds > 0 THEN
	nErrorID := iErrorDriveAds;
ELSIF iErrorDriveCAN > 0 THEN
	nErrorID := iErrorDriveCAN;
ELSIF iErrorEncAds > 0 THEN
	nErrorID := iErrorEncAds;
ELSE
	nErrorID := iErrorEncCAN;
END_IF

END_FUNCTION_BLOCK

// ---- POUs/FB_AxisRead70x1.TcPOU
FUNCTION_BLOCK FB_AxisRead70x1
VAR_INPUT
	bExecute: BOOL;
	bReset: BOOL;
	stDriveRef: ST_DriveRef;
END_VAR
VAR_IN_OUT
	stConfig: ST_AxisParams;
	Axis: AXIS_REF;
END_VAR
VAR_OUTPUT
	bBusy: BOOL;
	bError: BOOL;
	iAdsErrId: UINT;
	iCANopenErrId: UINT;
END_VAR
VAR
	fbReadMaxCurrent: FB_CoERead_ByDriveRef;
	nIndMaxCurrent: WORD;
	fbReadHoldingCurrent: FB_CoERead_ByDriveRef;
	nIndHoldingCurrent: WORD;
	fbReadVoltage: FB_CoERead_ByDriveRef;
	nIndVoltage: WORD;
	fbReadResistance: FB_CoERead_ByDriveRef;
	nIndResistance: WORD;
	fbReadEmf: FB_CoERead_ByDriveRef;
	nIndEmf: WORD;
	fbReadFullSteps: FB_CoERead_ByDriveRef;
	nIndFullSteps: WORD;
	fbReadSpeedRange: FB_CoERead_ByDriveRef;
	nIndSpeedRange: WORD;
END_VAR

// File auto-generated! Take care editing!
// Clears errors and allows a new read
IF bReset THEN
	bExecute := FALSE;
	bReset := FALSE;
END_IF
nIndMaxCurrent := 16#8010;
fbReadMaxCurrent(bExecute:=bExecute,
	stDriveRef:=stDriveRef,
	nindex:=nIndMaxCurrent,
	nSubIndex:=16#01,
	pDstBuf:=ADR(stConfig.max_current),
	cbBufLen:=SIZEOF(stConfig.max_current));
nIndHoldingCurrent := 16#8010;
fbReadHoldingCurrent(bExecute:=bExecute,
	stDriveRef:=stDriveRef,
	nindex:=nIndHoldingCurrent,
	nSubIndex:=16#02,
	pDstBuf:=ADR(stConfig.holding_current),
	cbBufLen:=SIZEOF(stConfig.holding_current));
nIndVoltage := 16#8010;
fbReadVoltage(bExecute:=bExecute,
	stDriveRef:=stDriveRef,
	nindex:=nIndVoltage,
	nSubIndex:=16#03,
	pDstBuf:=ADR(stConfig.voltage),
	cbBufLen:=SIZEOF(stConfig.voltage));
nIndResistance := 16#8010;
fbReadResistance(bExecute:=bExecute,
	stDriveRef:=stDriveRef,
	nindex:=nIndResistance,
	nSubIndex:=16#04,
	pDstBuf:=ADR(stConfig.resistance),
	cbBufLen:=SIZEOF(stConfig.resistance));
nIndEmf := 16#8010;
fbReadEmf(bExecute:=bExecute,
	stDriveRef:=stDriveRef,
	nindex:=nIndEmf,
	nSubIndex:=16#05,
	pDstBuf:=ADR(stConfig.emf),
	cbBufLen:=SIZEOF(stConfig.emf));
nIndFullSteps := 16#8010;
fbReadFullSteps(bExecute:=bExecute,
	stDriveRef:=stDriveRef,
	nindex:=nIndFullSteps,
	nSubIndex:=16#06,
	pDstBuf:=ADR(stConfig.full_steps),
	cbBufLen:=SIZEOF(stConfig.full_steps));
nIndSpeedRange := 16#8012;
fbReadSpeedRange(bExecute:=bExecute,
	stDriveRef:=stDriveRef,
	nindex:=nIndSpeedRange,
	nSubIndex:=16#05,
	pDstBuf:=ADR(stConfig.speed_range),
	cbBufLen:=SIZEOF(stConfig.speed_range));
bBusy := fbReadMaxCurrent.bBusy OR fbReadHoldingCurrent.bBusy OR fbReadVoltage.bBusy OR fbReadResistance.bBusy OR fbReadEmf.bBusy OR fbReadFullSteps.bBusy OR fbReadSpeedRange.bBusy;
bError := fbReadMaxCurrent.bError OR fbReadHoldingCurrent.bError OR fbReadVoltage.bError OR fbReadResistance.bError OR fbReadEmf.bError OR fbReadFullSteps.bError OR fbReadSpeedRange.bError;
IF NOT bError THEN
	iAdsErrId := 0;
ELSIF fbReadMaxCurrent.iAdsErrId > 0 THEN
	iAdsErrId := fbReadMaxCurrent.iAdsErrId;
ELSIF fbReadHoldingCurrent.iAdsErrId > 0 THEN
	iAdsErrId := fbReadHoldingCurrent.iAdsErrId;
ELSIF fbReadVoltage.iAdsErrId > 0 THEN
	iAdsErrId := fbReadVoltage.iAdsErrId;
ELSIF fbReadResistance.iAdsErrId > 0 THEN
	iAdsErrId := fbReadResistance.iAdsErrId;
ELSIF fbReadEmf.iAdsErrId > 0 THEN
	iAdsErrId := fbReadEmf.iAdsErrId;
ELSIF fbReadFullSteps.iAdsErrId > 0 THEN
	iAdsErrId := fbReadFullSteps.iAdsErrId;
ELSIF fbReadSpeedRange.iAdsErrId > 0 THEN
	iAdsErrId := fbReadSpeedRange.iAdsErrId;
END_IF
IF NOT bError THEN
	iCANopenErrId := 0;
ELSIF fbReadMaxCurrent.iCANopenErrId > 0 THEN
	iCANopenErrId := fbReadMaxCurrent.iCANopenErrId;
ELSIF fbReadHoldingCurrent.iCANopenErrId > 0 THEN
	iCANopenErrId := fbReadHoldingCurrent.iCANopenErrId;
ELSIF fbReadVoltage.iCANopenErrId > 0 THEN
	iCANopenErrId := fbReadVoltage.iCANopenErrId;
ELSIF fbReadResistance.iCANopenErrId > 0 THEN
	iCANopenErrId := fbReadResistance.iCANopenErrId;
ELSIF fbReadEmf.iCANopenErrId > 0 THEN
	iCANopenErrId := fbReadEmf.iCANopenErrId;
ELSIF fbReadFullSteps.iCANopenErrId > 0 THEN
	iCANopenErrId := fbReadFullSteps.iCANopenErrId;
ELSIF fbReadSpeedRange.iCANopenErrId > 0 THEN
	iCANopenErrId := fbReadSpeedRange.iCANopenErrId;
END_IF

END_FUNCTION_BLOCK

// ---- POUs/FB_AxisRead5042.TcPOU
FUNCTION_BLOCK FB_AxisRead5042
VAR_INPUT
	bExecute: BOOL;
	bReset: BOOL;
	stDriveRef: ST_DriveRef;
END_VAR
VAR_IN_OUT
	stConfig: ST_AxisParams;
	Axis: AXIS_REF;
END_VAR
VAR_OUTPUT
	bBusy: BOOL;
	bError: BOOL;
	iAdsErrId: UINT;
	iCANopenErrId: UINT;
END_VAR
VAR
	fbReadEncSupply: FB_CoERead_ByDriveRef;
	nIndEncSupply: WORD;
	fbReadEncClock: FB_CoERead_ByDriveRef;
	nIndEncClock: WORD;
	fbReadEncMultiBits: FB_CoERead_ByDriveRef;
	nIndEncMultiBits: WORD;
	fbReadEncSingleBits: FB_CoERead_ByDriveRef;
	nIndEncSingleBits: WORD;
END_VAR

// File auto-generated! Take care editing!
// Clears errors and allows a new read
IF bReset THEN
	bExecute := FALSE;
	bReset := FALSE;
END_IF
nIndEncSupply := 16#8008;
fbReadEncSupply(bExecute:=bExecute,
	stDriveRef:=stDriveRef,
	nindex:=nIndEncSupply,
	nSubIndex:=16#12,
	pDstBuf:=ADR(stConfig.enc_supply),
	cbBufLen:=SIZEOF(stConfig.enc_supply));
CASE stDriveRef.nDriveNo OF
	1:
		nIndEncClock := 16#8008;
	2:
		nIndEncClock := 16#8018;
END_CASE
fbReadEncClock(bExecute:=bExecute,
	stDriveRef:=stDriveRef,
	nindex:=nIndEncClock,
	nSubIndex:=16#13,
	pDstBuf:=ADR(stConfig.enc_clock),
	cbBufLen:=SIZEOF(stConfig.enc_clock));
CASE stDriveRef.nDriveNo OF
	1:
		nIndEncMultiBits := 16#8008;
	2:
		nIndEncMultiBits := 16#8018;
END_CASE
fbReadEncMultiBits(bExecute:=bExecute,
	stDriveRef:=stDriveRef,
	nindex:=nIndEncMultiBits,
	nSubIndex:=16#15,
	pDstBuf:=ADR(stConfig.enc_multi_bits),
	cbBufLen:=SIZEOF(stConfig.enc_multi_bits));
CASE stDriveRef.nDriveNo OF
	1:
		nIndEncSingleBits := 16#8008;
	2:
		nIndEncSingleBits := 16#8018;
END_CASE
fbReadEncSingleBits(bExecute:=bExecute,
	stDriveRef:=stDriveRef,
	nindex:=nIndEncSingleBits,
	nSubIndex:=16#16,
	pDstBuf:=ADR(stConfig.enc_single_bits),
	cbBufLen:=SIZEOF(stConfig.enc_single_bits));
bBusy := fbReadEncSupply.bBusy OR fbReadEncClock.bBusy OR fbReadEncMultiBits.bBusy OR fbReadEncSingleBits.bBusy;
bError := fbReadEncSupply.bError OR fbReadEncClock.bError OR fbReadEncMultiBits.bError OR fbReadEncSingleBits.bError;
IF NOT bError THEN
	iAdsErrId := 0;
ELSIF fbReadEncSupply.iAdsErrId > 0 THEN
	iAdsErrId := fbReadEncSupply.iAdsErrId;
ELSIF fbReadEncClock.iAdsErrId > 0 THEN
	iAdsErrId := fbReadEncClock.iAdsErrId;
ELSIF fbReadEncMultiBits.iAdsErrId > 0 THEN
	iAdsErrId := fbReadEncMultiBits.iAdsErrId;
ELSIF fbReadEncSingleBits.iAdsErrId > 0 THEN
	iAdsErrId := fbReadEncSingleBits.iAdsErrId;
END_IF
IF NOT bError THEN
	iCANopenErrId := 0;
ELSIF fbReadEncSupply.iCANopenErrId > 0 THEN
	iCANopenErrId := fbReadEncSupply.iCANopenErrId;
ELSIF fbReadEncClock.iCANopenErrId > 0 THEN
	iCANopenErrId := fbReadEncClock.iCANopenErrId;
ELSIF fbReadEncMultiBits.iCANopenErrId > 0 THEN
	iCANopenErrId := fbReadEncMultiBits.iCANopenErrId;
ELSIF fbReadEncSingleBits.iCANopenErrId > 0 THEN
	iCANopenErrId := fbReadEncSingleBits.iCANopenErrId;
END_IF

END_FUNCTION_BLOCK

// ---- POUs/FB_AxisWriteParams.TcPOU
FUNCTION_BLOCK FB_AxisWriteParams
VAR_INPUT
	bExecute: BOOL;
	bReset: BOOL;
	stConfig: ST_AxisParams;
	stHardware: ST_AxisHardware;
END_VAR
VAR_IN_OUT
	Axis: AXIS_REF;
END_VAR
VAR_OUTPUT
	bInitPreOp: BOOL;
	bDone: BOOL;
	bBusy: BOOL;
	bError: BOOL;
	nErrorID: UDINT;
END_VAR
VAR
	bDoWrite: BOOL;
	fbNCWrite: FB_AxisWriteNC;
	fbCoEWrite: FB_AxisWriteCoE;
	fbPrepWrite: FB_AxisSetSlaveState;
	fbInitState: FB_AxisSetSlaveState;
	fbPreOpState: FB_AxisSetSlaveState;
END_VAR

// Do not write unless axis is disabled. Leave TRUE after done to avoid resetting errors, etc.
bDoWrite := bExecute AND (Axis.Status.MotionState = MC_AXISSTATE_DISABLED OR bDone);
// Move to PREOP to prepare for writing
fbPrepWrite(bExecute:=bDoWrite,
	stHardware:=stHardware,
	reqState:=EC_DEVICE_STATE_PREOP);
// The first time we're here, report that we've set to PREOP so master can move to OP
IF fbPrepWrite.bDone AND NOT fbPrepWrite.bError THEN
	bInitPreOP := TRUE;
END_IF
// Do the write
fbNCWrite(bExecute:=fbPrepWrite.bDone AND NOT fbPrepWrite.bError,
	bReset:=bReset,
	stConfig:=stConfig,
	Axis:=Axis);
fbCoEWrite(bExecute:=fbNCWrite.bExecute,
	bReset:=bReset,
	stHardware:=stHardware,
	stConfig:=stConfig,
	Axis:=Axis);
// Move to INIT and back to PRE-OP for params that need a full restart
fbInitState(bExecute:=fbNCWrite.bDone AND NOT fbNCWrite.bError AND fbCoEWrite.bBusy AND NOT fbCoEWrite.bError,
	stHardware:=stHardware,
	reqState:=EC_DEVICE_STATE_INIT);
fbPreOpState(bExecute:=fbInitState.bDone AND NOT fbInitState.bError,
	stHardware:=stHardware,
	reqSTate:=EC_DEVICE_STATE_PREOP);
bDone := fbPreOpState.bDone;
bBusy := fbNCWrite.bBusy OR fbCoEWrite.bBusy OR fbPrepWrite.bBusy OR fbInitState.bBusy OR fbPreOpState.bBusy;
bError := fbNCWrite.bError OR fbCoEWrite.bError OR fbPrepWrite.bError OR fbInitState.bError OR fbPreOpState.bError;
IF fbNCWrite.nErrorID > 0 THEN
	nErrorID := fbNCWrite.nErrorID;
ELSIF fbCoeWrite.nErrorID > 0 THEN
	nErrorID := fbCoEWrite.nErrorID;
ELSIF fbPrepWrite.nErrId > 0 THEN
	nErrorID := fbPrepWrite.nErrId;
ELSIF fbInitSTate.nErrId > 0 THEN
	nErrorID := fbInitState.nErrId;
ELSE
	nErrorID := fbPreOpState.nErrId;
END_IF

END_FUNCTION_BLOCK

// ---- POUs/FB_AxisWriteNC.TcPOU
FUNCTION_BLOCK FB_AxisWriteNC
VAR_INPUT
	bExecute: BOOL;
	bReset: BOOL;
END_VAR
VAR_IN_OUT
	stConfig: ST_AxisParams;
	Axis: AXIS_REF;
END_VAR
VAR_OUTPUT
	bDone: BOOL;
	bBusy: BOOL;
	bError: BOOL;
	nErrorID: UDINT;
END_VAR
VAR
	fbWriteRefVel: MC_WriteParameter;
	fbWriteMaxVel: MC_WriteParameter;
	fbWriteMaxAcc: MC_WriteParameter;
	fbWriteMaxDec: MC_WriteParameter;
	fbWriteDefAcc: MC_WriteParameter;
	fbWriteDefDec: MC_WriteParameter;
	fbWriteDefJerk: MC_WriteParameter;
	fbWriteHomeSearch: MC_WriteParameter;
	fbWriteHomeSync: MC_WriteParameter;
	fbWriteManFast: MC_WriteParameter;
	fbWriteManSlow: MC_WriteParameter;
	fbWriteEnableMinSoftLimit: MC_WriteBoolParameter;
	fbWriteEnableMaxSoftLimit: MC_WriteBoolParameter;
	fbWriteMinSoftLimit: MC_WriteParameter;
	fbWriteMaxSoftLimit: MC_WriteParameter;
	fbWriteMaxPosLagValue: MC_WriteParameter;
	fbWriteMaxPosLagFilterTime: MC_WriteParameter;
	fbWriteDeadTime: MC_WriteParameter;
	fbWriteEncScale: MC_WriteParameter;
	fbWriteEncOffset: MC_WriteParameter;
	fbWriteEncInvert: MC_WriteBoolParameter;
	fbWriteMotInvert: MC_WriteBoolParameter;
END_VAR

// File auto-generated! Take care editing!
// Clears errors and allows a new read
IF bReset THEN
	bExecute := FALSE;
	bReset := FALSE;
END_IF
fbWriteRefVel(Execute:=bExecute,
	ParameterNumber:=MC_AxisParameter.AxisRefVeloOnRefOutput,
	Value:=stConfig.ref_vel,
	Axis:=Axis);
fbWriteMaxVel(Execute:=bExecute,
	ParameterNumber:=MC_AxisParameter.AxisMaxVelocity,
	Value:=stConfig.max_vel,
	Axis:=Axis);
fbWriteMaxAcc(Execute:=bExecute,
	ParameterNumber:=MC_AxisParameter.MaxAccelerationSystem,
	Value:=stConfig.max_acc,
	Axis:=Axis);
fbWriteMaxDec(Execute:=bExecute,
	ParameterNumber:=MC_AxisParameter.MaxDecelerationSystem,
	Value:=stConfig.max_dec,
	Axis:=Axis);
fbWriteDefAcc(Execute:=bExecute,
	ParameterNumber:=MC_AxisParameter.AxisAcc,
	Value:=stConfig.def_acc,
	Axis:=Axis);
fbWriteDefDec(Execute:=bExecute,
	ParameterNumber:=MC_AxisParameter.AxisDec,
	Value:=stConfig.def_dec,
	Axis:=Axis);
fbWriteDefJerk(Execute:=bExecute,
	ParameterNumber:=MC_AxisParameter.AxisJerk,
	Value:=stConfig.def_jerk,
	Axis:=Axis);
fbWriteHomeSearch(Execute:=bExecute,
	ParameterNumber:=MC_AxisParameter.AxisCalibrationVelocityForward,
	Value:=stConfig.home_search,
	Axis:=Axis);
fbWriteHomeSync(Execute:=bExecute,
	ParameterNumber:=MC_AxisParameter.AxisCalibrationVelocityBackward,
	Value:=stConfig.home_sync,
	Axis:=Axis);
fbWriteManFast(Execute:=bExecute,
	ParameterNumber:=MC_AxisParameter.AxisManualVelocityFast,
	Value:=stConfig.man_fast,
	Axis:=Axis);
fbWriteManSlow(Execute:=bExecute,
	ParameterNumber:=MC_AxisParameter.AxisManualVelocitySlow,
	Value:=stConfig.man_slow,
	Axis:=Axis);
fbWriteEnableMinSoftLimit(Execute:=bExecute,
	ParameterNumber:=MC_AxisParameter.EnableLimitNeg,
	Value:=stConfig.enable_min_soft_limit,
	Axis:=Axis);
fbWriteEnableMaxSoftLimit(Execute:=bExecute,
	ParameterNumber:=MC_AxisParameter.EnableLimitPos,
	Value:=stConfig.enable_max_soft_limit,
	Axis:=Axis);
fbWriteMinSoftLimit(Execute:=bExecute,
	ParameterNumber:=MC_AxisParameter.SWLimitNeg,
	Value:=stConfig.min_soft_limit,
	Axis:=Axis);
fbWriteMaxSoftLimit(Execute:=bExecute,
	ParameterNumber:=MC_AxisParameter.SWLimitPos,
	Value:=stConfig.max_soft_limit,
	Axis:=Axis);
fbWriteMaxPosLagValue(Execute:=bExecute,
	ParameterNumber:=MC_AxisParameter.MaxPositionLag,
	Value:=stConfig.max_pos_lag_value,
	Axis:=Axis);
fbWriteMaxPosLagFilterTime(Execute:=bExecute,
	ParameterNumber:=MC_AxisParameter.AxisMaxPosLagFilterTime,
	Value:=stConfig.max_pos_lag_filter_time,
	Axis:=Axis);
fbWriteDeadTime(Execute:=bExecute,
	ParameterNumber:=MC_AxisParameter.AxisDelayTimeVeloPosition,
	Value:=stConfig.dead_time,
	Axis:=Axis);
fbWriteEncScale(Execute:=bExecute,
	ParameterNumber:=MC_AxisParameter.AxisEncoderScalingFactor,
	Value:=stConfig.enc_scale,
	Axis:=Axis);
fbWriteEncOffset(Execute:=bExecute,
	ParameterNumber:=MC_AxisParameter.AxisEncoderOffset,
	Value:=stConfig.enc_offset,
	Axis:=Axis);
fbWriteEncInvert(Execute:=bExecute,
	ParameterNumber:=MC_AxisParameter.AxisEncoderDirectionInverse,
	Value:=stConfig.enc_invert,
	Axis:=Axis);
fbWriteMotInvert(Execute:=bExecute,
	ParameterNumber:=MC_AxisParameter.AxisMotorDirectionInverse,
	Value:=stConfig.mot_invert,
	Axis:=Axis);
bDone := fbWriteRefVel.Done AND fbWriteMaxVel.Done AND fbWriteMaxAcc.Done AND fbWriteMaxDec.Done AND fbWriteDefAcc.Done AND fbWriteDefDec.Done AND fbWriteDefJerk.Done AND fbWriteHomeSearch.Done AND fbWriteHomeSync.Done AND fbWriteManFast.Done AND fbWriteManSlow.Done AND fbWriteEnableMinSoftLimit.Done AND fbWriteEnableMaxSoftLimit.Done AND fbWriteMinSoftLimit.Done AND fbWriteMaxSoftLimit.Done AND fbWriteMaxPosLagValue.Done AND fbWriteMaxPosLagFilterTime.Done AND fbWriteDeadTime.Done AND fbWriteEncScale.Done AND fbWriteEncOffset.Done AND fbWriteEncInvert.Done AND fbWriteMotInvert.Done;
bBusy := fbWriteRefVel.Busy OR fbWriteMaxVel.Busy OR fbWriteMaxAcc.Busy OR fbWriteMaxDec.Busy OR fbWriteDefAcc.Busy OR fbWriteDefDec.Busy OR fbWriteDefJerk.Busy OR fbWriteHomeSearch.Busy OR fbWriteHomeSync.Busy OR fbWriteManFast.Busy OR fbWriteManSlow.Busy OR fbWriteEnableMinSoftLimit.Busy OR fbWriteEnableMaxSoftLimit.Busy OR fbWriteMinSoftLimit.Busy OR fbWriteMaxSoftLimit.Busy OR fbWriteMaxPosLagValue.Busy OR fbWriteMaxPosLagFilterTime.Busy OR fbWriteDeadTime.Busy OR fbWriteEncScale.Busy OR fbWriteEncOffset.Busy OR fbWriteEncInvert.Busy OR fbWriteMotInvert.Busy;
bError := fbWriteRefVel.Error OR fbWriteMaxVel.Error OR fbWriteMaxAcc.Error OR fbWriteMaxDec.Error OR fbWriteDefAcc.Error OR fbWriteDefDec.Error OR fbWriteDefJerk.Error OR fbWriteHomeSearch.Error OR fbWriteHomeSync.Error OR fbWriteManFast.Error OR fbWriteManSlow.Error OR fbWriteEnableMinSoftLimit.Error OR fbWriteEnableMaxSoftLimit.Error OR fbWriteMinSoftLimit.Error OR fbWriteMaxSoftLimit.Error OR fbWriteMaxPosLagValue.Error OR fbWriteMaxPosLagFilterTime.Error OR fbWriteDeadTime.Error OR fbWriteEncScale.Error OR fbWriteEncOffset.Error OR fbWriteEncInvert.Error OR fbWriteMotInvert.Error;
IF NOT bError THEN
	nErrorID := 0;
ELSIF fbWriteRefVel.ErrorID > 0 THEN
	nErrorID := fbWriteRefVel.ErrorID;
ELSIF fbWriteMaxVel.ErrorID > 0 THEN
	nErrorID := fbWriteMaxVel.ErrorID;
ELSIF fbWriteMaxAcc.ErrorID > 0 THEN
	nErrorID := fbWriteMaxAcc.ErrorID;
ELSIF fbWriteMaxDec.ErrorID > 0 THEN
	nErrorID := fbWriteMaxDec.ErrorID;
ELSIF fbWriteDefAcc.ErrorID > 0 THEN
	nErrorID := fbWriteDefAcc.ErrorID;
ELSIF fbWriteDefDec.ErrorID > 0 THEN
	nErrorID := fbWriteDefDec.ErrorID;
ELSIF fbWriteDefJerk.ErrorID > 0 THEN
	nErrorID := fbWriteDefJerk.ErrorID;
ELSIF fbWriteHomeSearch.ErrorID > 0 THEN
	nErrorID := fbWriteHomeSearch.ErrorID;
ELSIF fbWriteHomeSync.ErrorID > 0 THEN
	nErrorID := fbWriteHomeSync.ErrorID;
ELSIF fbWriteManFast.ErrorID > 0 THEN
	nErrorID := fbWriteManFast.ErrorID;
ELSIF fbWriteManSlow.ErrorID > 0 THEN
	nErrorID := fbWriteManSlow.ErrorID;
ELSIF fbWriteEnableMinSoftLimit.ErrorID > 0 THEN
	nErrorID := fbWriteEnableMinSoftLimit.ErrorID;
ELSIF fbWriteEnableMaxSoftLimit.ErrorID > 0 THEN
	nErrorID := fbWriteEnableMaxSoftLimit.ErrorID;
ELSIF fbWriteMinSoftLimit.ErrorID > 0 THEN
	nErrorID := fbWriteMinSoftLimit.ErrorID;
ELSIF fbWriteMaxSoftLimit.ErrorID > 0 THEN
	nErrorID := fbWriteMaxSoftLimit.ErrorID;
ELSIF fbWriteMaxPosLagValue.ErrorID > 0 THEN
	nErrorID := fbWriteMaxPosLagValue.ErrorID;
ELSIF fbWriteMaxPosLagFilterTime.ErrorID > 0 THEN
	nErrorID := fbWriteMaxPosLagFilterTime.ErrorID;
ELSIF fbWriteDeadTime.ErrorID > 0 THEN
	nErrorID := fbWriteDeadTime.ErrorID;
ELSIF fbWriteEncScale.ErrorID > 0 THEN
	nErrorID := fbWriteEncScale.ErrorID;
ELSIF fbWriteEncOffset.ErrorID > 0 THEN
	nErrorID := fbWriteEncOffset.ErrorID;
ELSIF fbWriteEncInvert.ErrorID > 0 THEN
	nErrorID := fbWriteEncInvert.ErrorID;
ELSIF fbWriteMotInvert.ErrorID > 0 THEN
	nErrorID := fbWriteMotInvert.ErrorID;
END_IF

END_FUNCTION_BLOCK

// ---- POUs/FB_AxisWriteCoE.TcPOU
FUNCTION_BLOCK FB_AxisWriteCoE
VAR_INPUT
	bExecute: BOOL;
	bReset: BOOL;
	stHardware: ST_AxisHardware;
END_VAR
VAR_IN_OUT
	stConfig: ST_AxisParams;
	Axis: AXIS_REF;
END_VAR
VAR_OUTPUT
	bDone: BOOL;
	bBusy: BOOL;
	bError: BOOL;
	nErrorID: UDINT;
END_VAR
VAR
	fbWrite70x1: FB_AxisWrite70x1;
	fbWrite5042: FB_AxisWrite5042;
	bBusyDrive: BOOL;
	bBusyEnc: BOOL;
	bErrorDrive: BOOL;
	bErrorEnc: BOOL;
	iErrorDriveADS: UDINT;
	iErrorEncADS: UDINT;
	iErrorDriveCAN: UDINT;
	iErrorEncCAN: UDINT;
END_VAR

CASE stHardware.drive_type OF
	0:
		bBusyDrive := FALSE;
		bErrorDrive := FALSE;
		iErrorDriveAds := 0;
		iErrorDriveCAN := 0;
	7031, 7041:
		fbWrite70x1(bExecute:=bExecute,
			bReset:=bReset,
			stDriveRef:=stHardware.drive_ref,
			stConfig:=stConfig,
			Axis:=Axis,
			bBusy=>bBusyDrive,
			bError=>bErrorDrive,
			iAdsErrId=>iErrorDriveAds,
			iCANopenErrId=>iErrorDriveCAN);
	ELSE
		bBusyDrive := FALSE;
		bErrorDrive := TRUE;
		iErrorDriveAds := 1;
		iErrorDriveCAN := 0;
END_CASE
CASE stHardware.enc_type OF
	0:
		bBusyEnc := FALSE;
		bErrorEnc := FALSE;
		iErrorEncAds := 0;
		iErrorEncCAN := 0;
	5042:
		fbWrite5042(bExecute:=bExecute,
			bReset:=bReset,
			stDriveRef:=stHardware.enc_ref,
			stConfig:=stConfig,
			Axis:=Axis,
			bBusy=>bBusyEnc,
			bError=>bErrorEnc,
			iAdsErrId=>iErrorEncAds,
			iCANopenErrId=>iErrorEncCAN);
	ELSE
		bBusyEnc := FALSE;
		bErrorEnc := TRUE;
		iErrorEncAds := 1;
		iErrorEncCAN := 0;
END_CASE
bBusy := bBusyDrive OR bBusyEnc;
bDone := bExecute AND NOT bBusy;
bError := bErrorDrive OR bErrorEnc;
IF iErrorDriveAds > 0 THEN
	nErrorID := iErrorDriveAds;
ELSIF iErrorDriveCAN > 0 THEN
	nErrorID := iErrorDriveCAN;
ELSIF iErrorEncAds > 0 THEN
	nErrorID := iErrorEncAds;
ELSE
	nErrorID := iErrorEncCAN;
END_IF

END_FUNCTION_BLOCK

// ---- POUs/FB_AxisWrite70x1.TcPOU
FUNCTION_BLOCK FB_AxisWrite70x1
VAR_INPUT
	bExecute: BOOL;
	bReset: BOOL;
	stDriveRef: ST_DriveRef;
	stConfig: ST_AxisParams;
END_VAR
VAR_IN_OUT
	Axis: AXIS_REF;
END_VAR
VAR_OUTPUT
	bBusy: BOOL;
	bError: BOOL;
	iAdsErrId: UINT;
	iCANopenErrId: UINT;
END_VAR
VAR
	fbWriteMaxCurrent: FB_CoEWrite_ByDriveRef;
	nIndMaxCurrent: WORD;
	fbWriteHoldingCurrent: FB_CoEWrite_ByDriveRef;
	nIndHoldingCurrent: WORD;
	fbWriteVoltage: FB_CoEWrite_ByDriveRef;
	nIndVoltage: WORD;
	fbWriteResistance: FB_CoEWrite_ByDriveRef;
	nIndResistance: WORD;
	fbWriteEmf: FB_CoEWrite_ByDriveRef;
	nIndEmf: WORD;
	fbWriteFullSteps: FB_CoEWrite_ByDriveRef;
	nIndFullSteps: WORD;
	fbWriteSpeedRange: FB_CoEWrite_ByDriveRef;
	nIndSpeedRange: WORD;
END_VAR

// File auto-generated! Take care editing!
// Clears errors and allows a new read
IF bReset THEN
	bExecute := FALSE;
	bReset := FALSE;
END_IF
nIndMaxCurrent := 16#8010;
fbWriteMaxCurrent(bExecute:=bExecute,
	stDriveRef:=stDriveRef,
	nindex:=nIndMaxCurrent,
	nSubIndex:=16#01,
	pSrcBuf:=ADR(stConfig.max_current),
	cbBufLen:=SIZEOF(stConfig.max_current));
nIndHoldingCurrent := 16#8010;
fbWriteHoldingCurrent(bExecute:=bExecute,
	stDriveRef:=stDriveRef,
	nindex:=nIndHoldingCurrent,
	nSubIndex:=16#02,
	pSrcBuf:=ADR(stConfig.holding_current),
	cbBufLen:=SIZEOF(stConfig.holding_current));
nIndVoltage := 16#8010;
fbWriteVoltage(bExecute:=bExecute,
	stDriveRef:=stDriveRef,
	nindex:=nIndVoltage,
	nSubIndex:=16#03,
	pSrcBuf:=ADR(stConfig.voltage),
	cbBufLen:=SIZEOF(stConfig.voltage));
nIndResistance := 16#8010;
fbWriteResistance(bExecute:=bExecute,
	stDriveRef:=stDriveRef,
	nindex:=nIndResistance,
	nSubIndex:=16#04,
	pSrcBuf:=ADR(stConfig.resistance),
	cbBufLen:=SIZEOF(stConfig.resistance));
nIndEmf := 16#8010;
fbWriteEmf(bExecute:=bExecute,
	stDriveRef:=stDriveRef,
	nindex:=nIndEmf,
	nSubIndex:=16#05,
	pSrcBuf:=ADR(stConfig.emf),
	cbBufLen:=SIZEOF(stConfig.emf));
nIndFullSteps := 16#8010;
fbWriteFullSteps(bExecute:=bExecute,
	stDriveRef:=stDriveRef,
	nindex:=nIndFullSteps,
	nSubIndex:=16#06,
	pSrcBuf:=ADR(stConfig.full_steps),
	cbBufLen:=SIZEOF(stConfig.full_steps));
nIndSpeedRange := 16#8012;
fbWriteSpeedRange(bExecute:=bExecute,
	stDriveRef:=stDriveRef,
	nindex:=nIndSpeedRange,
	nSubIndex:=16#05,
	pSrcBuf:=ADR(stConfig.speed_range),
	cbBufLen:=SIZEOF(stConfig.speed_range));
bBusy := fbWriteMaxCurrent.bBusy OR fbWriteHoldingCurrent.bBusy OR fbWriteVoltage.bBusy OR fbWriteResistance.bBusy OR fbWriteEmf.bBusy OR fbWriteFullSteps.bBusy OR fbWriteSpeedRange.bBusy;
bError := fbWriteMaxCurrent.bError OR fbWriteHoldingCurrent.bError OR fbWriteVoltage.bError OR fbWriteResistance.bError OR fbWriteEmf.bError OR fbWriteFullSteps.bError OR fbWriteSpeedRange.bError;
IF NOT bError THEN
	iAdsErrId := 0;
ELSIF fbWriteMaxCurrent.iAdsErrId > 0 THEN
	iAdsErrId := fbWriteMaxCurrent.iAdsErrId;
ELSIF fbWriteHoldingCurrent.iAdsErrId > 0 THEN
	iAdsErrId := fbWriteHoldingCurrent.iAdsErrId;
ELSIF fbWriteVoltage.iAdsErrId > 0 THEN
	iAdsErrId := fbWriteVoltage.iAdsErrId;
ELSIF fbWriteResistance.iAdsErrId > 0 THEN
	iAdsErrId := fbWriteResistance.iAdsErrId;
ELSIF fbWriteEmf.iAdsErrId > 0 THEN
	iAdsErrId := fbWriteEmf.iAdsErrId;
ELSIF fbWriteFullSteps.iAdsErrId > 0 THEN
	iAdsErrId := fbWriteFullSteps.iAdsErrId;
ELSIF fbWriteSpeedRange.iAdsErrId > 0 THEN
	iAdsErrId := fbWriteSpeedRange.iAdsErrId;
END_IF
IF NOT bError THEN
	iCANopenErrId := 0;
ELSIF fbWriteMaxCurrent.iCANopenErrId > 0 THEN
	iCANopenErrId := fbWriteMaxCurrent.iCANopenErrId;
ELSIF fbWriteHoldingCurrent.iCANopenErrId > 0 THEN
	iCANopenErrId := fbWriteHoldingCurrent.iCANopenErrId;
ELSIF fbWriteVoltage.iCANopenErrId > 0 THEN
	iCANopenErrId := fbWriteVoltage.iCANopenErrId;
ELSIF fbWriteResistance.iCANopenErrId > 0 THEN
	iCANopenErrId := fbWriteResistance.iCANopenErrId;
ELSIF fbWriteEmf.iCANopenErrId > 0 THEN
	iCANopenErrId := fbWriteEmf.iCANopenErrId;
ELSIF fbWriteFullSteps.iCANopenErrId > 0 THEN
	iCANopenErrId := fbWriteFullSteps.iCANopenErrId;
ELSIF fbWriteSpeedRange.iCANopenErrId > 0 THEN
	iCANopenErrId := fbWriteSpeedRange.iCANopenErrId;
END_IF

END_FUNCTION_BLOCK

// ---- POUs/FB_AxisWrite5042.TcPOU
FUNCTION_BLOCK FB_AxisWrite5042
VAR_INPUT
	bExecute: BOOL;
	bReset: BOOL;
	stDriveRef: ST_DriveRef;
	stConfig: ST_AxisParams;
END_VAR
VAR_IN_OUT
	Axis: AXIS_REF;
END_VAR
VAR_OUTPUT
	bBusy: BOOL;
	bError: BOOL;
	iAdsErrId: UINT;
	iCANopenErrId: UINT;
END_VAR
VAR
	fbWriteEncSupply: FB_CoEWrite_ByDriveRef;
	nIndEncSupply: WORD;
	fbWriteEncClock: FB_CoEWrite_ByDriveRef;
	nIndEncClock: WORD;
	fbWriteEncMultiBits: FB_CoEWrite_ByDriveRef;
	nIndEncMultiBits: WORD;
	fbWriteEncSingleBits: FB_CoEWrite_ByDriveRef;
	nIndEncSingleBits: WORD;
END_VAR

// File auto-generated! Take care editing!
// Clears errors and allows a new read
IF bReset THEN
	bExecute := FALSE;
	bReset := FALSE;
END_IF
nIndEncSupply := 16#8008;
fbWriteEncSupply(bExecute:=bExecute,
	stDriveRef:=stDriveRef,
	nindex:=nIndEncSupply,
	nSubIndex:=16#12,
	pSrcBuf:=ADR(stConfig.enc_supply),
	cbBufLen:=SIZEOF(stConfig.enc_supply));
CASE stDriveRef.nDriveNo OF
	1:
		nIndEncClock := 16#8008;
	2:
		nIndEncClock := 16#8018;
END_CASE
fbWriteEncClock(bExecute:=bExecute,
	stDriveRef:=stDriveRef,
	nindex:=nIndEncClock,
	nSubIndex:=16#13,
	pSrcBuf:=ADR(stConfig.enc_clock),
	cbBufLen:=SIZEOF(stConfig.enc_clock));
CASE stDriveRef.nDriveNo OF
	1:
		nIndEncMultiBits := 16#8008;
	2:
		nIndEncMultiBits := 16#8018;
END_CASE
fbWriteEncMultiBits(bExecute:=bExecute,
	stDriveRef:=stDriveRef,
	nindex:=nIndEncMultiBits,
	nSubIndex:=16#15,
	pSrcBuf:=ADR(stConfig.enc_multi_bits),
	cbBufLen:=SIZEOF(stConfig.enc_multi_bits));
CASE stDriveRef.nDriveNo OF
	1:
		nIndEncSingleBits := 16#8008;
	2:
		nIndEncSingleBits := 16#8018;
END_CASE
fbWriteEncSingleBits(bExecute:=bExecute,
	stDriveRef:=stDriveRef,
	nindex:=nIndEncSingleBits,
	nSubIndex:=16#16,
	pSrcBuf:=ADR(stConfig.enc_single_bits),
	cbBufLen:=SIZEOF(stConfig.enc_single_bits));
bBusy := fbWriteEncSupply.bBusy OR fbWriteEncClock.bBusy OR fbWriteEncMultiBits.bBusy OR fbWriteEncSingleBits.bBusy;
bError := fbWriteEncSupply.bError OR fbWriteEncClock.bError OR fbWriteEncMultiBits.bError OR fbWriteEncSingleBits.bError;
IF NOT bError THEN
	iAdsErrId := 0;
ELSIF fbWriteEncSupply.iAdsErrId > 0 THEN
	iAdsErrId := fbWriteEncSupply.iAdsErrId;
ELSIF fbWriteEncClock.iAdsErrId > 0 THEN
	iAdsErrId := fbWriteEncClock.iAdsErrId;
ELSIF fbWriteEncMultiBits.iAdsErrId > 0 THEN
	iAdsErrId := fbWriteEncMultiBits.iAdsErrId;
ELSIF fbWriteEncSingleBits.iAdsErrId > 0 THEN
	iAdsErrId := fbWriteEncSingleBits.iAdsErrId;
END_IF
IF NOT bError THEN
	iCANopenErrId := 0;
ELSIF fbWriteEncSupply.iCANopenErrId > 0 THEN
	iCANopenErrId := fbWriteEncSupply.iCANopenErrId;
ELSIF fbWriteEncClock.iCANopenErrId > 0 THEN
	iCANopenErrId := fbWriteEncClock.iCANopenErrId;
ELSIF fbWriteEncMultiBits.iCANopenErrId > 0 THEN
	iCANopenErrId := fbWriteEncMultiBits.iCANopenErrId;
ELSIF fbWriteEncSingleBits.iCANopenErrId > 0 THEN
	iCANopenErrId := fbWriteEncSingleBits.iCANopenErrId;
END_IF

END_FUNCTION_BLOCK

// ---- POUs/FB_AxisSetSlaveState.TcPOU
FUNCTION_BLOCK FB_AxisSetSlaveState
VAR_INPUT
	bExecute: BOOL;
	stHardware: ST_AxisHardware;
	reqState: WORD;
END_VAR
VAR_OUTPUT
	bDone: BOOL;
	bBusy: BOOL;
	bError: BOOL;
	nErrId: UDINT;
	currStateDrive: ST_EcSlaveState;
	currStateEnc: ST_EcSlaveState;
END_VAR
VAR
	fbDriveState: FB_EcSetSlaveState;
	fbEncState: FB_EcSetSlaveState;
	bBusyDrive: BOOL;
	bBusyEnc: BOOL;
	bErrorDrive: BOOL;
	bErrorEnc: BOOL;
	nErrIdDrive: UDINT;
	nErrIdEnc: UDINT;
END_VAR

// Transition terminals if they exist
IF stHardware.drive_type > 0 THEN
	fbDriveState(sNetID:=stHardware.drive_ref.sNetId,
		nSlaveAddr:=stHardware.drive_ref.nSlaveAddr,
		bExecute:=bExecute,
		reqState:=reqState,
		bBusy=>bBusyDrive,
		bError=>bErrorDrive,
		nErrId=>nErrIdDrive,
		currState=>currStateDrive);
ELSE
	bBusyDrive := FALSE;
	bErrorDrive := FALSE;
	nErrIdDrive := 0;
END_IF
IF stHardware.enc_type > 0 THEN
	fbEncState(sNetID:=stHardware.enc_ref.sNetId,
		nSlaveAddr:=stHardware.enc_ref.nSlaveAddr,
		bExecute:=bExecute,
		reqState:=reqState,
		bBusy=>bBusyDrive,
		bError=>bErrorDrive,
		nErrId=>nErrIdDrive,
		currState=>currStateEnc);
ELSE
	bBusyEnc := FALSE;
	bErrorEnc := FALSE;
	nErrIdDrive := 0;
END_IF
bBusy := bBusyDrive OR bBusyEnc;
bDone := bExecute AND NOT bBusy;
bError := bErrorDrive OR bErrorEnc;
IF nErrIdDrive > 0 THEN
	nErrId := nErrIdDrive;
ELSE
	nErrId := nErrIdEnc;
END_IF

END_FUNCTION_BLOCK
